Staubli VAL3: Align.pgx

program Align(tool x_tTool, bool& x_bOK)
  local point l_pPoint
  local point l_pPoint1
  local bool l_bSame
begin
  //-----------------------------------------------------------------------
  //Header begin
  //Description of program
  //  工具对齐
  //Input parameters
  //  tool x_tTool:工具值
  //Output paramaters
  //  bool x_bOK:是否对齐
  //Example
  //  call Align(tool,bOK)
  //History
  //  Creation : 2012-06-11 - PF.Zhong
  //Header end
  //-----------------------------------------------------------------------
  resetMotion()
  x_bOK=false
  link(l_pPoint,world)
  link(l_pPoint1,world)
  l_pPoint=here(x_tTool,world)
  l_pPoint1.trsf=align(l_pPoint.trsf,world.trsf)
  call ComparePoint(l_pPoint,l_pPoint1,l_bSame)
  if !l_bSame
    movej(l_pPoint1,x_tTool,mNomSpeed)
    waitEndMove()
    delay(0.1)
    l_pPoint=here(x_tTool,world)
    call ComparePoint(l_pPoint,l_pPoint1,l_bSame)
    if l_bSame
      x_bOK=true
    else
      x_bOK=false
    endIf
  else
    x_bOK=true
  endIf
end
